(* IEC 61131-3 sources: automationbase/test/Supervisions, 3 files *)

(* ---- SupervisionAssert.st ---- *)
USING AxUnit.ResultFunctions;
USING Simatic.Ax.AutomationBase;
USING System.Strings;

NAMESPACE AutomationBase.Tests

    /// Assert für SupervisionError Enum
    FUNCTION PUBLIC EqualSupervisionError
        VAR_INPUT
            expected : SupervisionError;
            actual : SupervisionError;
            {CallerFilePath}
            file : WSTRING[1024];
            {CallerLineNumber}
            line : INT;
        END_VAR
        VAR_TEMP
            message : STRING[254];
        END_VAR

        IF expected = actual THEN
            axunit_Succeed();
        ELSE
            message := 'Expected SupervisionError to be ';
            CASE expected OF
                SupervisionError#NO_ERROR:
                    message := Concat(message, 'NO_ERROR');
                SupervisionError#TIMEOUT:
                    message := Concat(message, 'TIMEOUT');
            END_CASE;
            message := Concat(message, ' but was ');
            CASE actual OF
                SupervisionError#NO_ERROR:
                    message := Concat(message, 'NO_ERROR');
                SupervisionError#TIMEOUT:
                    message := Concat(message, 'TIMEOUT');
            END_CASE;
            axunit_Fail(message, file, line);
        END_IF;
    END_FUNCTION

    /// Assert für SupervisionBehavior Enum
    FUNCTION PUBLIC EqualSupervisionBehavior
        VAR_INPUT
            expected : SupervisionBehavior;
            actual : SupervisionBehavior;
            {CallerFilePath}
            file : WSTRING[1024];
            {CallerLineNumber}
            line : INT;
        END_VAR
        VAR_TEMP
            message : STRING[254];
        END_VAR

        IF expected = actual THEN
            axunit_Succeed();
        ELSE
            message := 'Expected SupervisionBehavior to be ';
            CASE expected OF
                SupervisionBehavior#Action:
                    message := Concat(message, 'Action');
                SupervisionBehavior#Reaction:
                    message := Concat(message, 'Reaction');
            END_CASE;
            message := Concat(message, ' but was ');
            CASE actual OF
                SupervisionBehavior#Action:
                    message := Concat(message, 'Action');
                SupervisionBehavior#Reaction:
                    message := Concat(message, 'Reaction');
            END_CASE;
            axunit_Fail(message, file, line);
        END_IF;
    END_FUNCTION

END_NAMESPACE

(* ---- SupervisionIntegrationTest.st ---- *)
USING AxUnit.Assert;
USING AxUnit.Mocking;
USING Simatic.Ax.AutomationBase;
USING AutomationBase.Tests;

NAMESPACE AutomationBase.Tests

    {TestFixture}
    CLASS SupervisionIntegrationTest
        VAR
            // Stateless copies für jeden Test
            _cylinder_supervision, _cylinder_supervisionStateless : Supervision;
            _motor_supervision, _motor_supervisionStateless : Supervision;
            _two_stage_action, _two_stage_actionStateless : Supervision;
            _two_stage_reaction, _two_stage_reactionStateless : Supervision;
        END_VAR

        //=============================================================================
        // SETUP
        //=============================================================================

        {TestSetup}
        METHOD PUBLIC TestSetup
            // Kopiere stateless Instanzen für jeden Test
            _cylinder_supervision := _cylinder_supervisionStateless;
            _motor_supervision := _motor_supervisionStateless;
            _two_stage_action := _two_stage_actionStateless;
            _two_stage_reaction := _two_stage_reactionStateless;
        END_METHOD

        //=============================================================================
        // INTEGRATIONSTESTS FÜR PNEUMATIKZYLINDER
        //=============================================================================

        {Test}
        METHOD PUBLIC Test_PneumaticCylinder_SuccessfulExtension
            VAR_TEMP
                cylinder_extended : BOOL;
                cylinder_retracted : BOOL;
            END_VAR

            // Arrange - Zylinder eingefahren
            Mock(NAME_OF(System.Timer.OnDelay), NAME_OF(Simatic.Ax.Mocks.OnDelayMock_false));
            cylinder_retracted := TRUE;
            cylinder_extended := FALSE;
            _cylinder_supervision.timeout := T#100ms;
            _cylinder_supervision.behavior := SupervisionBehavior#Action;

            // Act - Starte Ausfahren
            _cylinder_supervision.Start();

            // Simuliere Zylinderfahrt (nach 5 Zyklen erreicht)
            THIS.SimulateCylinderExtension(
                supervision := _cylinder_supervision,
                cycles_until_extended := 5,
                cylinder_extended := cylinder_extended
            );

            // Assert
            Equal(expected := TRUE, actual := _cylinder_supervision.IsCompleted());
            Equal(expected := FALSE, actual := _cylinder_supervision.HasError());
        END_METHOD

        {Test}
        METHOD PUBLIC Test_PneumaticCylinder_BlockedExtension
            VAR_TEMP
                cylinder_extended : BOOL;
            END_VAR

            // Arrange - Zylinder blockiert
            Mock(NAME_OF(System.Timer.OnDelay), NAME_OF(Simatic.Ax.Mocks.OnDelayMock_true));
            cylinder_extended := FALSE;
            _cylinder_supervision.timeout := T#10ms;
            _cylinder_supervision.behavior := SupervisionBehavior#Action;

            // Act - Starte Ausfahren, aber Zylinder bleibt blockiert
            _cylinder_supervision.Start();

            // Zylinder bewegt sich nicht - Timer läuft ab
            _cylinder_supervision.Execute(signal := cylinder_extended);

            // Assert
            Equal(expected := TRUE, actual := _cylinder_supervision.HasError());
            EqualSupervisionError(expected := SupervisionError#TIMEOUT, actual := _cylinder_supervision.GetError());
        END_METHOD

        {Test}
        METHOD PUBLIC Test_PneumaticCylinder_RetractAfterExtend
            VAR_TEMP
                cylinder_extended : BOOL;
            END_VAR

            // Test: Ausfahren und dann Einfahren
            Mock(NAME_OF(System.Timer.OnDelay), NAME_OF(Simatic.Ax.Mocks.OnDelayMock_false));

            // Phase 1: Ausfahren
            cylinder_extended := FALSE;
            _cylinder_supervision.timeout := T#100ms;
            _cylinder_supervision.behavior := SupervisionBehavior#Action;
            _cylinder_supervision.Start();
            THIS.SimulateCylinderExtension(
                supervision := _cylinder_supervision,
                cycles_until_extended := 5,
                cylinder_extended := cylinder_extended
            );
            Equal(expected := TRUE, actual := _cylinder_supervision.IsCompleted());

            // Phase 2: Einfahren
            _cylinder_supervision.Reset();
            _cylinder_supervision.behavior := SupervisionBehavior#Reaction;
            _cylinder_supervision.Start();
            THIS.SimulateCylinderRetraction(
                supervision := _cylinder_supervision,
                cycles_until_retracted := 5,
                cylinder_extended := cylinder_extended
            );
            Equal(expected := TRUE, actual := _cylinder_supervision.IsCompleted());
        END_METHOD

        //=============================================================================
        // INTEGRATIONSTESTS FÜR MOTORSTART
        //=============================================================================

        {Test}
        METHOD PUBLIC Test_Motor_SuccessfulStart
            VAR_TEMP
                motor_running : BOOL;
            END_VAR

            // Arrange
            Mock(NAME_OF(System.Timer.OnDelay), NAME_OF(Simatic.Ax.Mocks.OnDelayMock_false));
            motor_running := FALSE;
            _motor_supervision.timeout := T#50ms;
            _motor_supervision.behavior := SupervisionBehavior#Action;

            // Act - Motor starten
            _motor_supervision.Start();
            THIS.SimulateMotorStart(
                supervision := _motor_supervision,
                cycles_until_running := 3,
                motor_running := motor_running
            );

            // Assert
            Equal(expected := TRUE, actual := _motor_supervision.IsCompleted());
        END_METHOD

        {Test}
        METHOD PUBLIC Test_Motor_FailedStart
            VAR_TEMP
                motor_running : BOOL;
            END_VAR

            // Arrange - Motor startet nicht
            Mock(NAME_OF(System.Timer.OnDelay), NAME_OF(Simatic.Ax.Mocks.OnDelayMock_true));
            motor_running := FALSE;
            _motor_supervision.timeout := T#10ms;
            _motor_supervision.behavior := SupervisionBehavior#Action;

            // Act - Versuch Motor zu starten
            _motor_supervision.Start();
            _motor_supervision.Execute(signal := motor_running);

            // Assert
            Equal(expected := TRUE, actual := _motor_supervision.HasError());
        END_METHOD

        //=============================================================================
        // INTEGRATIONSTESTS FÜR ZWEISTUFIGE ÜBERWACHUNG
        //=============================================================================

        {Test}
        METHOD PUBLIC Test_TwoStage_SuccessfulMovement
            VAR_TEMP
                position_left_start : BOOL;
                position_at_target : BOOL;
            END_VAR

            // Test: Bewegung mit Aktions- und Reaktionsüberwachung
            Mock(NAME_OF(System.Timer.OnDelay), NAME_OF(Simatic.Ax.Mocks.OnDelayMock_false));

            // Arrange
            position_left_start := FALSE;
            position_at_target := FALSE;
            _two_stage_action.timeout := T#50ms;
            _two_stage_action.behavior := SupervisionBehavior#Action;
            _two_stage_reaction.timeout := T#100ms;
            _two_stage_reaction.behavior := SupervisionBehavior#Action;

            // Act Phase 1: Aktionsüberwachung (Bewegung beginnt)
            _two_stage_action.Start();
            THIS.SimulateMovementStart(
                supervision := _two_stage_action,
                cycles_until_started := 3,
                position_left_start := position_left_start
            );
            Equal(expected := TRUE, actual := _two_stage_action.IsCompleted());

            // Act Phase 2: Reaktionsüberwachung (Bewegung endet)
            _two_stage_reaction.Start();
            THIS.SimulateMovementEnd(
                supervision := _two_stage_reaction,
                cycles_until_target := 5,
                position_at_target := position_at_target
            );

            // Assert
            Equal(expected := TRUE, actual := _two_stage_reaction.IsCompleted());
        END_METHOD

        {Test}
        METHOD PUBLIC Test_TwoStage_FailsInActionPhase
            VAR_TEMP
                position_left_start : BOOL;
            END_VAR

            // Test: Bewegung beginnt nicht
            Mock(NAME_OF(System.Timer.OnDelay), NAME_OF(Simatic.Ax.Mocks.OnDelayMock_true));

            // Arrange
            position_left_start := FALSE;
            _two_stage_action.timeout := T#10ms;
            _two_stage_action.behavior := SupervisionBehavior#Action;

            // Act - Bewegung beginnt nicht
            _two_stage_action.Start();
            _two_stage_action.Execute(signal := position_left_start);

            // Assert
            Equal(expected := TRUE, actual := _two_stage_action.HasError());
        END_METHOD

        {Test}
        METHOD PUBLIC Test_TwoStage_FailsInReactionPhase
            VAR_TEMP
                position_left_start : BOOL;
                position_at_target : BOOL;
            END_VAR

            // Test: Bewegung beginnt, aber erreicht Ziel nicht
            Mock(NAME_OF(System.Timer.OnDelay), NAME_OF(Simatic.Ax.Mocks.OnDelayMock_false));

            // Arrange
            position_left_start := FALSE;
            position_at_target := FALSE;
            _two_stage_action.timeout := T#50ms;
            _two_stage_action.behavior := SupervisionBehavior#Action;
            _two_stage_reaction.timeout := T#10ms;
            _two_stage_reaction.behavior := SupervisionBehavior#Action;

            // Act Phase 1: Bewegung beginnt erfolgreich
            _two_stage_action.Start();
            THIS.SimulateMovementStart(
                supervision := _two_stage_action,
                cycles_until_started := 3,
                position_left_start := position_left_start
            );
            Equal(expected := TRUE, actual := _two_stage_action.IsCompleted());

            // Act Phase 2: Ziel wird nicht erreicht
            Mock(NAME_OF(System.Timer.OnDelay), NAME_OF(Simatic.Ax.Mocks.OnDelayMock_true));
            _two_stage_reaction.Start();
            _two_stage_reaction.Execute(signal := position_at_target);

            // Assert
            Equal(expected := TRUE, actual := _two_stage_reaction.HasError());
        END_METHOD

        //=============================================================================
        // HILFSMETHODEN FÜR SIMULATION
        //=============================================================================

        METHOD PRIVATE SimulateCylinderExtension
            VAR_IN_OUT
                supervision : Supervision;
                cylinder_extended : BOOL;
            END_VAR
            VAR_INPUT
                cycles_until_extended : INT;
            END_VAR
            VAR
                i : INT;
            END_VAR

            FOR i := 1 TO cycles_until_extended DO
                supervision.Execute(signal := cylinder_extended);
            END_FOR;

            // Zylinder erreicht Endposition
            cylinder_extended := TRUE;
            supervision.Execute(signal := cylinder_extended);
        END_METHOD

        METHOD PRIVATE SimulateCylinderRetraction
            VAR_IN_OUT
                supervision : Supervision;
                cylinder_extended : BOOL;
            END_VAR
            VAR_INPUT
                cycles_until_retracted : INT;
            END_VAR
            VAR
                i : INT;
            END_VAR

            FOR i := 1 TO cycles_until_retracted DO
                supervision.Execute(signal := cylinder_extended);
            END_FOR;

            // Zylinder erreicht Endposition
            cylinder_extended := FALSE;
            supervision.Execute(signal := cylinder_extended);
        END_METHOD

        METHOD PRIVATE SimulateMotorStart
            VAR_IN_OUT
                supervision : Supervision;
                motor_running : BOOL;
            END_VAR
            VAR_INPUT
                cycles_until_running : INT;
            END_VAR
            VAR
                i : INT;
            END_VAR

            FOR i := 1 TO cycles_until_running DO
                supervision.Execute(signal := motor_running);
            END_FOR;

            // Motor läuft
            motor_running := TRUE;
            supervision.Execute(signal := motor_running);
        END_METHOD

        METHOD PRIVATE SimulateMovementStart
            VAR_IN_OUT
                supervision : Supervision;
                position_left_start : BOOL;
            END_VAR
            VAR_INPUT
                cycles_until_started : INT;
            END_VAR
            VAR
                i : INT;
            END_VAR

            FOR i := 1 TO cycles_until_started DO
                supervision.Execute(signal := position_left_start);
            END_FOR;

            // Startposition verlassen
            position_left_start := TRUE;
            supervision.Execute(signal := position_left_start);
        END_METHOD

        METHOD PRIVATE SimulateMovementEnd
            VAR_IN_OUT
                supervision : Supervision;
                position_at_target : BOOL;
            END_VAR
            VAR_INPUT
                cycles_until_target : INT;
            END_VAR
            VAR
                i : INT;
            END_VAR

            FOR i := 1 TO cycles_until_target DO
                supervision.Execute(signal := position_at_target);
            END_FOR;

            // Zielposition erreicht
            position_at_target := TRUE;
            supervision.Execute(signal := position_at_target);
        END_METHOD

    END_CLASS

END_NAMESPACE

(* ---- SupervisionTest.st ---- *)
USING AxUnit.Assert;
USING AxUnit.Mocking;
USING Simatic.Ax.AutomationBase;
USING AutomationBase.Tests;

NAMESPACE AutomationBase.Tests

    {TestFixture}
    CLASS SupervisionTest
        VAR
            // Stateless copies für jeden Test
            _supervision, _supervisionStateless : Supervision;
        END_VAR

        //=============================================================================
        // SETUP
        //=============================================================================

        {TestSetup}
        METHOD PUBLIC TestSetup
            // Kopiere stateless Instanz für jeden Test
            _supervision := _supervisionStateless;

            // Konfiguration
            _supervision.timeout := T#100ms;
            _supervision.behavior := SupervisionBehavior#Action;
        END_METHOD

        //=============================================================================
        // TESTS FÜR ACTION-VERHALTEN (Signal muss TRUE werden)
        //=============================================================================

        {Test}
        METHOD PUBLIC Test_Action_SignalBecomesTrue_CompletesSuccessfully
            VAR_TEMP
                testSignal : BOOL;
            END_VAR

            // Arrange
            Mock(NAME_OF(System.Timer.OnDelay), NAME_OF(Simatic.Ax.Mocks.OnDelayMock_false));
            _supervision.behavior := SupervisionBehavior#Action;
            _supervision.Start();

            // Act - Signal wird TRUE
            testSignal := TRUE;
            _supervision.Execute(signal := testSignal);

            // Assert
            Equal(expected := TRUE, actual := _supervision.IsCompleted());
            Equal(expected := FALSE, actual := _supervision.HasError());
            Equal(expected := FALSE, actual := _supervision.IsActive());
        END_METHOD

        {Test}
        METHOD PUBLIC Test_Action_SignalStaysFalse_CausesTimeout
            VAR_TEMP
                testSignal : BOOL;
            END_VAR

            // Arrange
            Mock(NAME_OF(System.Timer.OnDelay), NAME_OF(Simatic.Ax.Mocks.OnDelayMock_true));
            _supervision.behavior := SupervisionBehavior#Action;
            _supervision.Start();

            // Act - Signal bleibt FALSE, Timer gibt TRUE zurück (Timeout)
            testSignal := FALSE;
            _supervision.Execute(signal := testSignal);

            // Assert
            Equal(expected := TRUE, actual := _supervision.HasError());
            EqualSupervisionError(expected := SupervisionError#TIMEOUT, actual := _supervision.GetError());
            Equal(expected := FALSE, actual := _supervision.IsActive());
            Equal(expected := FALSE, actual := _supervision.IsCompleted());
        END_METHOD

        {Test}
        METHOD PUBLIC Test_Action_SignalBecomesTrueBeforeTimeout_NoError
            VAR_TEMP
                testSignal : BOOL;
            END_VAR

            // Arrange
            Mock(NAME_OF(System.Timer.OnDelay), NAME_OF(Simatic.Ax.Mocks.OnDelayMock_false));
            _supervision.behavior := SupervisionBehavior#Action;
            _supervision.Start();

            // Act - Signal wird TRUE vor Timeout
            testSignal := FALSE;
            _supervision.Execute(signal := testSignal);
            testSignal := TRUE;
            _supervision.Execute(signal := testSignal);

            // Assert
            Equal(expected := FALSE, actual := _supervision.HasError());
            Equal(expected := TRUE, actual := _supervision.IsCompleted());
        END_METHOD

        //=============================================================================
        // TESTS FÜR REACTION-VERHALTEN (Signal muss FALSE werden)
        //=============================================================================

        {Test}
        METHOD PUBLIC Test_Reaction_SignalBecomesFalse_CompletesSuccessfully
            VAR_TEMP
                testSignal : BOOL;
            END_VAR

            // Arrange
            Mock(NAME_OF(System.Timer.OnDelay), NAME_OF(Simatic.Ax.Mocks.OnDelayMock_false));
            _supervision.behavior := SupervisionBehavior#Reaction;
            _supervision.Start();

            // Act - Signal wird FALSE
            testSignal := FALSE;
            _supervision.Execute(signal := testSignal);

            // Assert
            Equal(expected := TRUE, actual := _supervision.IsCompleted());
            Equal(expected := FALSE, actual := _supervision.HasError());
            Equal(expected := FALSE, actual := _supervision.IsActive());
        END_METHOD

        {Test}
        METHOD PUBLIC Test_Reaction_SignalStaysTrue_CausesTimeout
            VAR_TEMP
                testSignal : BOOL;
            END_VAR

            // Arrange
            Mock(NAME_OF(System.Timer.OnDelay), NAME_OF(Simatic.Ax.Mocks.OnDelayMock_true));
            _supervision.behavior := SupervisionBehavior#Reaction;
            _supervision.Start();

            // Act - Signal bleibt TRUE, Timer gibt TRUE zurück (Timeout)
            testSignal := TRUE;
            _supervision.Execute(signal := testSignal);

            // Assert
            Equal(expected := TRUE, actual := _supervision.HasError());
            EqualSupervisionError(expected := SupervisionError#TIMEOUT, actual := _supervision.GetError());
            Equal(expected := FALSE, actual := _supervision.IsActive());
        END_METHOD

        {Test}
        METHOD PUBLIC Test_Reaction_SignalBecomesFalseBeforeTimeout_NoError
            VAR_TEMP
                testSignal : BOOL;
            END_VAR

            // Arrange
            Mock(NAME_OF(System.Timer.OnDelay), NAME_OF(Simatic.Ax.Mocks.OnDelayMock_false));
            _supervision.behavior := SupervisionBehavior#Reaction;
            _supervision.Start();

            // Act - Signal wird FALSE vor Timeout
            testSignal := TRUE;
            _supervision.Execute(signal := testSignal);
            testSignal := FALSE;
            _supervision.Execute(signal := testSignal);

            // Assert
            Equal(expected := FALSE, actual := _supervision.HasError());
            Equal(expected := TRUE, actual := _supervision.IsCompleted());
        END_METHOD

        //=============================================================================
        // TESTS FÜR START/STOP/RESET
        //=============================================================================

        {Test}
        METHOD PUBLIC Test_Start_ActivatesSupervision
            // Act
            _supervision.Start();

            // Assert
            Equal(expected := TRUE, actual := _supervision.IsActive());
            Equal(expected := FALSE, actual := _supervision.IsCompleted());
            Equal(expected := FALSE, actual := _supervision.HasError());
        END_METHOD

        {Test}
        METHOD PUBLIC Test_Stop_DeactivatesSupervision
            // Arrange
            _supervision.Start();

            // Act
            _supervision.Stop();

            // Assert
            Equal(expected := FALSE, actual := _supervision.IsActive());
            Equal(expected := FALSE, actual := _supervision.HasError());
        END_METHOD

        {Test}
        METHOD PUBLIC Test_Reset_ClearsErrorAndStops
            VAR_TEMP
                testSignal : BOOL;
            END_VAR

            // Arrange
            Mock(NAME_OF(System.Timer.OnDelay), NAME_OF(Simatic.Ax.Mocks.OnDelayMock_true));
            _supervision.Start();
            testSignal := FALSE;
            _supervision.Execute(signal := testSignal);
            Equal(expected := TRUE, actual := _supervision.HasError());

            // Act
            _supervision.Reset();

            // Assert
            Equal(expected := FALSE, actual := _supervision.HasError());
            Equal(expected := FALSE, actual := _supervision.IsActive());
            EqualSupervisionError(expected := SupervisionError#NO_ERROR, actual := _supervision.GetError());
        END_METHOD

        {Test}
        METHOD PUBLIC Test_MultipleStarts_ResetsState
            VAR_TEMP
                testSignal : BOOL;
            END_VAR

            // Arrange
            Mock(NAME_OF(System.Timer.OnDelay), NAME_OF(Simatic.Ax.Mocks.OnDelayMock_false));
            _supervision.Start();
            testSignal := TRUE;
            _supervision.Execute(signal := testSignal);
            Equal(expected := TRUE, actual := _supervision.IsCompleted());

            // Act - Erneuter Start
            _supervision.Start();

            // Assert
            Equal(expected := TRUE, actual := _supervision.IsActive());
            Equal(expected := FALSE, actual := _supervision.IsCompleted());
            Equal(expected := FALSE, actual := _supervision.HasError());
        END_METHOD

        //=============================================================================
        // TESTS FÜR EDGE CASES
        //=============================================================================

        {Test}
        METHOD PUBLIC Test_ExecuteWithoutStart_DoesNothing
            VAR_TEMP
                testSignal : BOOL;
            END_VAR

            // Act - Execute ohne Start
            testSignal := TRUE;
            _supervision.Execute(signal := testSignal);

            // Assert
            Equal(expected := FALSE, actual := _supervision.IsActive());
            Equal(expected := FALSE, actual := _supervision.IsCompleted());
            Equal(expected := FALSE, actual := _supervision.HasError());
        END_METHOD

        {Test}
        METHOD PUBLIC Test_ExecuteAfterCompletion_DoesNotChangeState
            VAR_TEMP
                testSignal : BOOL;
            END_VAR

            // Arrange
            Mock(NAME_OF(System.Timer.OnDelay), NAME_OF(Simatic.Ax.Mocks.OnDelayMock_false));
            _supervision.Start();
            testSignal := TRUE;
            _supervision.Execute(signal := testSignal);
            Equal(expected := TRUE, actual := _supervision.IsCompleted());

            // Act - Weitere Execute-Aufrufe
            testSignal := FALSE;
            _supervision.Execute(signal := testSignal);

            // Assert - Zustand bleibt unverändert
            Equal(expected := TRUE, actual := _supervision.IsCompleted());
            Equal(expected := FALSE, actual := _supervision.HasError());
        END_METHOD

        {Test}
        METHOD PUBLIC Test_ExecuteAfterError_DoesNotChangeState
            VAR_TEMP
                testSignal : BOOL;
            END_VAR

            // Arrange - Erzeuge Timeout
            Mock(NAME_OF(System.Timer.OnDelay), NAME_OF(Simatic.Ax.Mocks.OnDelayMock_true));
            _supervision.Start();
            testSignal := FALSE;
            _supervision.Execute(signal := testSignal);
            Equal(expected := TRUE, actual := _supervision.HasError());

            // Act - Weitere Execute-Aufrufe
            testSignal := TRUE;
            _supervision.Execute(signal := testSignal);

            // Assert - Fehler bleibt bestehen
            Equal(expected := TRUE, actual := _supervision.HasError());
            Equal(expected := FALSE, actual := _supervision.IsCompleted());
        END_METHOD

        //=============================================================================
        // TESTS FÜR ZUSTANDSÜBERGÄNGE
        //=============================================================================

        {Test}
        METHOD PUBLIC Test_StateTransition_NotStarted_To_Active
            // Initial
            Equal(expected := FALSE, actual := _supervision.IsActive());

            // Start
            _supervision.Start();
            Equal(expected := TRUE, actual := _supervision.IsActive());
        END_METHOD

        {Test}
        METHOD PUBLIC Test_StateTransition_Active_To_Completed
            VAR_TEMP
                testSignal : BOOL;
            END_VAR

            // Arrange
            Mock(NAME_OF(System.Timer.OnDelay), NAME_OF(Simatic.Ax.Mocks.OnDelayMock_false));

            // Start
            _supervision.Start();
            Equal(expected := TRUE, actual := _supervision.IsActive());

            // Complete
            testSignal := TRUE;
            _supervision.Execute(signal := testSignal);
            Equal(expected := FALSE, actual := _supervision.IsActive());
            Equal(expected := TRUE, actual := _supervision.IsCompleted());
        END_METHOD

        {Test}
        METHOD PUBLIC Test_StateTransition_Active_To_Error
            VAR_TEMP
                testSignal : BOOL;
            END_VAR

            // Arrange
            Mock(NAME_OF(System.Timer.OnDelay), NAME_OF(Simatic.Ax.Mocks.OnDelayMock_true));

            // Start
            _supervision.Start();
            Equal(expected := TRUE, actual := _supervision.IsActive());

            // Timeout
            testSignal := FALSE;
            _supervision.Execute(signal := testSignal);
            Equal(expected := FALSE, actual := _supervision.IsActive());
            Equal(expected := TRUE, actual := _supervision.HasError());
        END_METHOD

    END_CLASS

END_NAMESPACE
